// TIA Portal V20 export
// export: Created 2025-12-01T14:57:43.1054253Z, ExportSetting None, DisplayName Totally Integrated Automation Portal, DisplayVersion V20 Update 3, DisplayName TIA Portal Openness, DisplayVersion V20 Update 3, DisplayName TIA Portal Version Control Interface, DisplayVersion V20 Update 3, DisplayName STEP 7 Professional, DisplayVersion V20 Update 3, DisplayName STEP 7 Safety, DisplayVersion V20 Update 2, DisplayName WinCC Basic/Comfort/Advanced, DisplayVersion V20 Update 3, DisplayName WinCC Professional, DisplayVersion V20 Update 3, DisplayName WinCC Unified, DisplayVersion V20 Update 3
DATA_BLOCK "DB927_PNIODiag_Data"   // DB927
{ S7_Optimized_Access := 'FALSE' }
// stored: AutoNumber false
   VAR RETAIN
      RED : Array[1..5] of Struct
         NODO : Array[1..256] of Struct
            had_failed : Bool;
            deactivated : Bool;
            reserved_10 : Bool;
            reserved_11 : Bool;
            reserved_12 : Bool;
            reserved_13 : Bool;
            reserved_14 : Bool;
            reserved_15 : Bool;
            OK : Bool;
            maintenance : Bool;
            faulty : Bool;
            failed : Bool;
            was_deactivated : Bool;
            DPV1 : Bool;
            was_under_maintenance : Bool;
            was_failed : Bool;
         END_STRUCT;
      END_STRUCT;
   END_VAR
BEGIN
END_DATA_BLOCK
